(*
SPDX-FileCopyrightText: Â© 2026 Oleksandr Tiutyk <trofimich@gmail.com>
SPDX-License-Identifier: MIT
License: https://opensource.org/license/mit
*)

(*!
<summary>Read-only contract for a digital output automation component.</summary>
<description>
Provides access to logical boolean output state, change detection and electrical contact configuration.
</description>
*)

INTERFACE IReadOnlyDigitalOutput EXTENDS TOF_Automation.IOutputLeafAutomationComponent

(*!
<summary>Indicates whether the current logical command differs from the last processed command.</summary>
<description>
ProcessOutput() acknowledges the current command even without an I/O binding.
</description>
*)
{attribute 'monitoring' := 'call'}
PROPERTY Changed : BOOL
GET
END_GET
END_PROPERTY

(*!
<summary>Gets electrical contact configuration.</summary>
*)
{attribute 'monitoring' := 'call'}
PROPERTY ContactType : CONTACT_TYPE
GET
END_GET
END_PROPERTY

(*!
<summary>Gets current evaluated logical state of the output signal.</summary>
*)
{attribute 'monitoring' := 'call'}
PROPERTY Value : BOOL
GET
END_GET
END_PROPERTY

END_INTERFACE

(* stored: Version 1.1.0.1
   Itf IReadOnlyDigitalOutput: Id {5d606187-b064-4d50-9ede-efa1febf93e9}
   Property Changed: Id {19d66a30-b4e7-4315-bc9b-36bffdc623cb}
   Get Get: Id {b3e13947-62e0-4bd3-86a4-fd7aaafe100e}
   Property ContactType: Id {ba70bd05-3243-4c30-8dab-160463eedd98}
   Get Get: Id {a5114882-2308-465f-a67a-8b781d0333af}
   Property Value: Id {901ff42a-ef4e-4a96-86b6-4b131bb3516d}
   Get Get: Id {f8e5fa2c-0123-46ac-b700-12f1d3b71cec} *)
